FUNCTION_BLOCK FB_TestProtocol EXTENDS FB_SocketClientProtocolBase
VAR_INPUT
	send_data : ST_SendDataFormat;
END_VAR
VAR_OUTPUT
	receive_data : ST_ReceiveDataFormat;
END_VAR
VAR
END_VAR

METHOD Parse : BOOL
IF SIZEOF(receive_data) = MEMCPY(ADR(receive_data), ADR(SUPER^.receive_data_buffer), SIZEOF(receive_data)) THEN
	Parse := TRUE;
END_IF
END_METHOD

PROPERTY received : BOOL
GET
VAR
	specified_size : UDINT;
END_VAR
specified_size := SIZEOF(receive_data);
received := SUPER^.receive_data_size = specified_size;
END_GET
END_PROPERTY

PROPERTY SendData : ST_CommunicationMetaData
GET
SendData.cbLen := SIZEOF(send_data);
SendData.pData := ADR(send_data);
END_GET
END_PROPERTY

END_FUNCTION_BLOCK

(* stored: Version 1.1.0.1, ProductVersion 3.1.4024.15
   POU FB_TestProtocol: Id {3c9ec079-52dc-40d5-bd05-b4062fa89375}, SpecialFunc None
   Method Parse: Id {8af2c580-c5e8-41a8-b779-bea6e4de146a}
   Property received: Id {f489726b-1376-41d8-900b-f60a890949fb}
   Get Get: Id {9fe03456-0e59-422c-8b47-08bdac5bf07d}
   Property SendData: Id {eed17491-b3ea-4268-ac9f-17a42bb3947b}
   Get Get: Id {7533733c-c3ea-4d4b-a6a5-f7c286120254} *)
